TYPE Room_Settings_TimeSettings :
STRUCT
	nOff		: UDINT := TIME_TO_UDINT(T#30S);
	nOn			: UDINT := TIME_TO_UDINT(T#30S);
END_STRUCT
END_TYPE

(* stored: Version 1.1.0.1
   DUT Room_Settings_TimeSettings: Id {a09af3f3-b6d2-4d22-a191-50ef57298cc4} *)
